FUNCTION_BLOCK FB_Skalowanie
VAR_INPUT
	Ymax: REAL;
	Xmax: REAL;
	Xmin: REAL;
	Ymin: REAL;
	X: REAL;
END_VAR
VAR_OUTPUT
	Y: REAL;
	bAlarmLo: BOOL;
	bALarmHi: BOOL;
END_VAR
VAR
	A: REAL;
	B: REAL;
END_VAR

IF X<=Xmin THEN
	
	Y:=Ymin;
	bAlarmLo:=TRUE;
	bALarmHi:=FALSE;

ELSIF X>=Xmax THEN
	
	Y:=Ymax;
	bAlarmLo:=FALSE;
	bALarmHi:=TRUE;

ELSE
	IF Xmax<> Xmin THEN
	
		A:=(Ymax-Ymin)/(Xmax-Xmin);
		B:=Ymax-A*Xmax;
		Y:=A*X+B;
		bAlarmLo:=FALSE;
		bALarmHi:=FALSE;
		
	ELSE
		
		Y:=Ymax;
		bAlarmLo:=TRUE;
		bALarmHi:=TRUE;
		
	END_IF;
END_IF;

END_FUNCTION_BLOCK

(* stored: Version 1.1.0.1, ProductVersion 3.1.4026.13, FileIdentifier 739913c66acbbd72eba817fa4cf61a323b60db37, FileSignature 0b83dd3f82630cb56b7460619e27b842edbde8e8880022b2719378c8feb7abc5b30d38d3efe9d7a15fb9efc96c52095f6bbf506e0fdb9035fe0b5aadb7ad382cf33ad715d57df7c320a56c706110ced67fde37c854dfbebec1ef7dfd58a5309b57678b625deb9a0a76528048df36aa06d5047caa66af257ce4171a87ea4915d8bf8fb75e446f01263ae07c519e8f3c2a628ce685279e424bae394b1f961d7ee1974f56c799589b0055d4865a419e676f9986023c1965d5003be37c254ddf6c5e80e1ca64b5b410ecfd7930fc10bcbc68642b4c9e2f4827ac87315d6278973533d81f853137066abbfd54f0ddec8c463051ba53ac19513d009877121c541171d5
   POU FB_Skalowanie: Id {ba0ad885-f70c-43d0-85ca-56862c232a02}, SpecialFunc None *)
